// Mitsubishi GX Works2 project: Final_Version   PLC: FX3G

// global labels: Global1
VAR_GLOBAL
  DayStartSwitch AT X007 : BOOL;
  NotInStockSwitch AT M41 : BOOL;
  DayLight AT Y007 : BOOL;
  IceMakeSwitch AT X001 : BOOL;
  AnalogInput1 AT D8280 : INT;
END_VAR
VAR_GLOBAL CONSTANT
  UpperBound_K10 : REAL := 10.0;
  LowerBound_K0 : REAL;
  PetelNeeded_K280 : REAL := 280.0;
  LemonNeeded_K455 : REAL := 455.0;
  StabilityNeeded_K105 : REAL := 105.0;
  GumiBearsNeeded_K28 : REAL := 28.0;
  PetelNeeded_K385 : REAL := 385.0;
  LemonNeeded_K665 : REAL := 665.0;
  StabilityNeeded_K210 : REAL := 210.0;
  GumiBearsNeeded_K70 : REAL := 70.0;
END_VAR
VAR_GLOBAL
  RegularGumiLight AT M42 : BOOL;
END_VAR
VAR_GLOBAL CONSTANT
  Regular_GumiGam_k5 : REAL := 5.0;
  Special_GumiGam_K6 : REAL := 6.0;
END_VAR
VAR_GLOBAL
  IceMakeLight AT Y000 : BOOL;
  IceMakeTimer AT TC1 : BOOL;
  DayFinishSwitch AT M11 : BOOL;
END_VAR
VAR_GLOBAL CONSTANT
  IceMakeCounter_K50 : INT := 50;
  CounterValue_K1 : INT := 1;
  K400_const : REAL := 400.0;
END_VAR
VAR_GLOBAL
  PossibleRegularGumi AT M43 : BOOL;
  SpecialGumiLight AT M45 : BOOL;
  IcePetelContainer_IceMake AT D1500 : REAL;
  IceLemonContainer_IceMake AT D2500 : REAL;
  SaveAnalog_1_Value AT D5100 : REAL;
  PetelStock AT D1100 : REAL;
  LemonStock AT D2100 : REAL;
  StabilityStock AT D3100 : REAL;
  GumiBearsStock AT D4100 : REAL;
  IceMakeCounter_Finish AT CS0 : BOOL;
  IceMakeTimer_Finish AT TS1 : BOOL;
  IceMakeCounter AT CC0 : BOOL;
END_VAR
VAR_GLOBAL CONSTANT
  IceMakeTimer_K50 : INT := 50;
END_VAR
VAR_GLOBAL
  PossibleSpecialGumi AT M44 : BOOL;
  CoolingSwitchX002 AT X002 : BOOL;
  CoolingContainerPetel AT D6000 : REAL;
  CoolingContainerLemon AT D6010 : REAL;
  CoolingTimerDone AT TS2 : BOOL;
  CoolingFinishedCounter AT CC7 : BOOL;
  CoolingLightY002 AT Y002 : BOOL;
  CoolingTimer AT TC2 : BOOL;
END_VAR
VAR_GLOBAL CONSTANT
  CoolingTimeValue : INT := 80;
END_VAR
VAR_GLOBAL
  TempIndicatorX003 AT X003 : BOOL;
END_VAR
VAR_GLOBAL CONSTANT
  NormalGumiBears : REAL := 28;
  PinukGumiBears : REAL := 70;
  ResetContainer : REAL;
END_VAR
VAR_GLOBAL
  MixingContainer AT D6030 : REAL;
END_VAR
VAR_GLOBAL CONSTANT
  BlinkingCounterNormal : REAL := 3;
END_VAR
VAR_GLOBAL
  BlinkingCounterChosen AT D6040 : REAL;
END_VAR
VAR_GLOBAL CONSTANT
  BlinkingCounterPinuk : REAL := 5;
END_VAR
VAR_GLOBAL
  BlinkingLight5 AT Y005 : BOOL;
END_VAR
VAR_GLOBAL CONSTANT
  BlinkingTimerValue : INT := 10;
END_VAR
VAR_GLOBAL
  BlinkingTimer1 AT TC24 : BOOL;
  blinkingTriger AT M32 : BOOL;
  BlinkingTimerDone1 AT TS24 : BOOL;
  BlinkingTimeIsUp AT CS10 : BOOL;
  BlinkingLight6 AT Y006 : BOOL;
  BlinkingTimer2 AT TC25 : BOOL;
  BlinkingTimerDone2 AT TS25 : BOOL;
  BlinkingTimesUpCounter AT CC10 : BOOL;
  Stock AT D6050 : REAL;
END_VAR
VAR_GLOBAL CONSTANT
  FinishedPackage : REAL := 1;
END_VAR
VAR_GLOBAL
  AnalogOut AT D8282 : INT;
  EmergencyStop AT X005 : BOOL;
END_VAR
VAR_GLOBAL CONSTANT
  K40_const : REAL := 40;
  IcePetelRegular_K350 : REAL := 350;
  IcePetelPinuk_K560 : REAL := 560;
  IceLemonRegular_K490 : REAL := 490;
  IceLemonPinuk_K700 : REAL := 700;
END_VAR
VAR_GLOBAL
  InValidInput AT Y010 : BOOL;
  CoolingFinishedCounter_Finish AT CS7 : BOOL;
END_VAR

// task Task_01 (event TRUE, interval 0, priority 31): POU_01

PROGRAM POU_01
(* structured ladder/FBD written out as ST: instructions are called as NAME(EN, inputs, outputs); _pN, _eN, _tN stand for wires *)
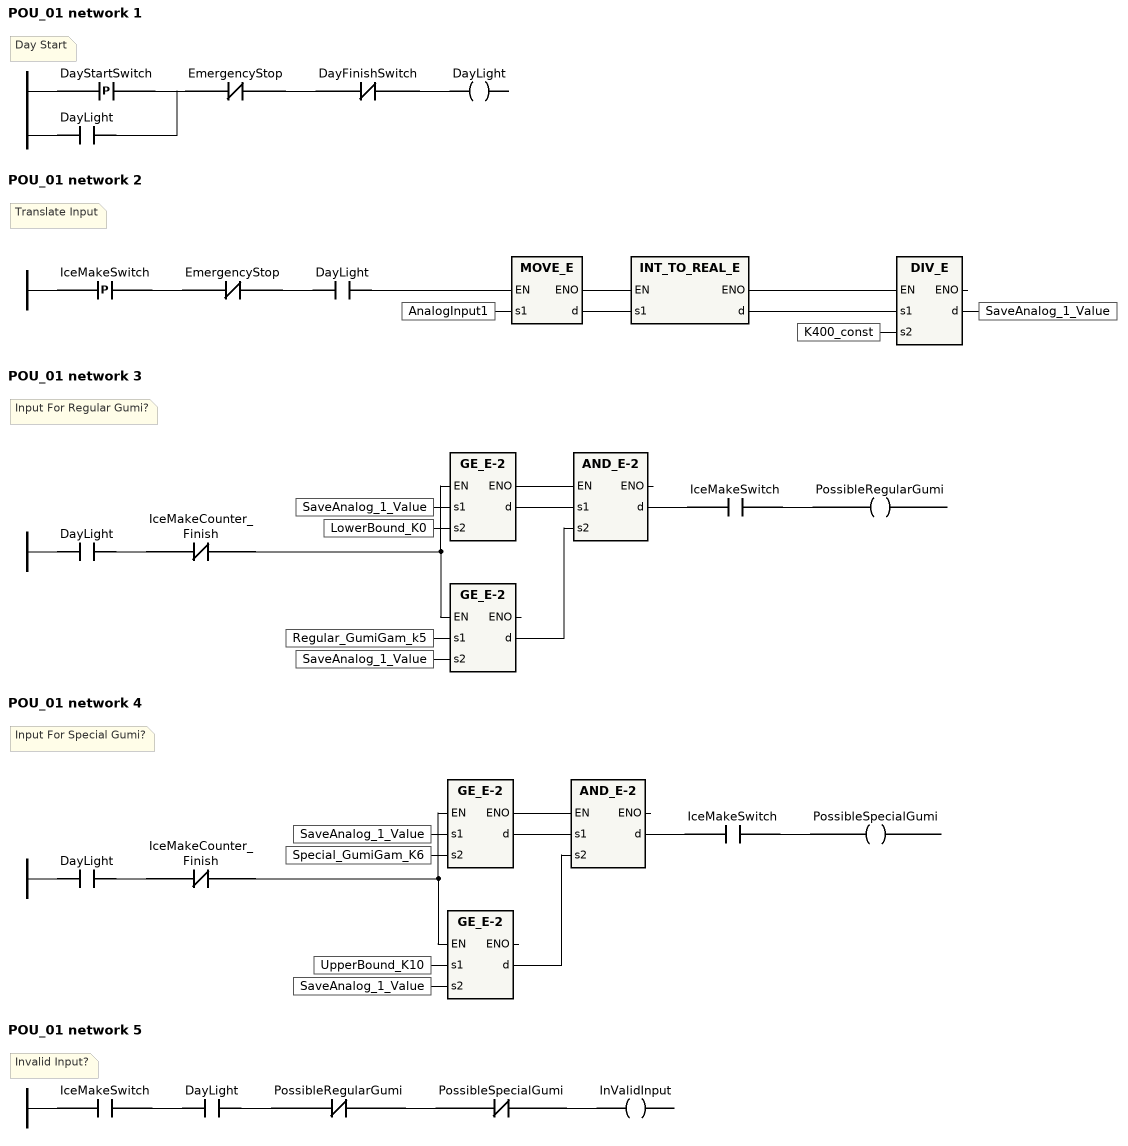
(* network 1 *)
(* Day Start *)
DayLight := ((LDP(TRUE, DayStartSwitch) OR DayLight) AND NOT EmergencyStop) AND NOT DayFinishSwitch;
(* network 2 *)
(* Translate Input *)
_e2 := MOVE_E(LDP(TRUE, IceMakeSwitch) AND NOT EmergencyStop AND DayLight, AnalogInput1, _t1);
_e4 := INT_TO_REAL_E(_e2, _t1, _t3);
DIV_E(_e4, _t3, K400_const, SaveAnalog_1_Value);
(* network 3 *)
(* Input For Regular Gumi? *)
_p1 := DayLight AND NOT IceMakeCounter_Finish;
_e3 := GE_E(_p1, SaveAnalog_1_Value, LowerBound_K0, _t2);
GE_E(_p1, Regular_GumiGam_k5, SaveAnalog_1_Value, _t4);
AND_E(_e3, _t2, _t4, _t5);
PossibleRegularGumi := _t5 AND IceMakeSwitch;
(* network 4 *)
(* Input For Special Gumi? *)
_p1 := DayLight AND NOT IceMakeCounter_Finish;
_e3 := GE_E(_p1, SaveAnalog_1_Value, Special_GumiGam_K6, _t2);
GE_E(_p1, UpperBound_K10, SaveAnalog_1_Value, _t4);
AND_E(_e3, _t2, _t4, _t5);
PossibleSpecialGumi := _t5 AND IceMakeSwitch;
(* network 5 *)
(* Invalid Input? *)
InValidInput := IceMakeSwitch AND DayLight AND NOT PossibleRegularGumi AND NOT PossibleSpecialGumi;
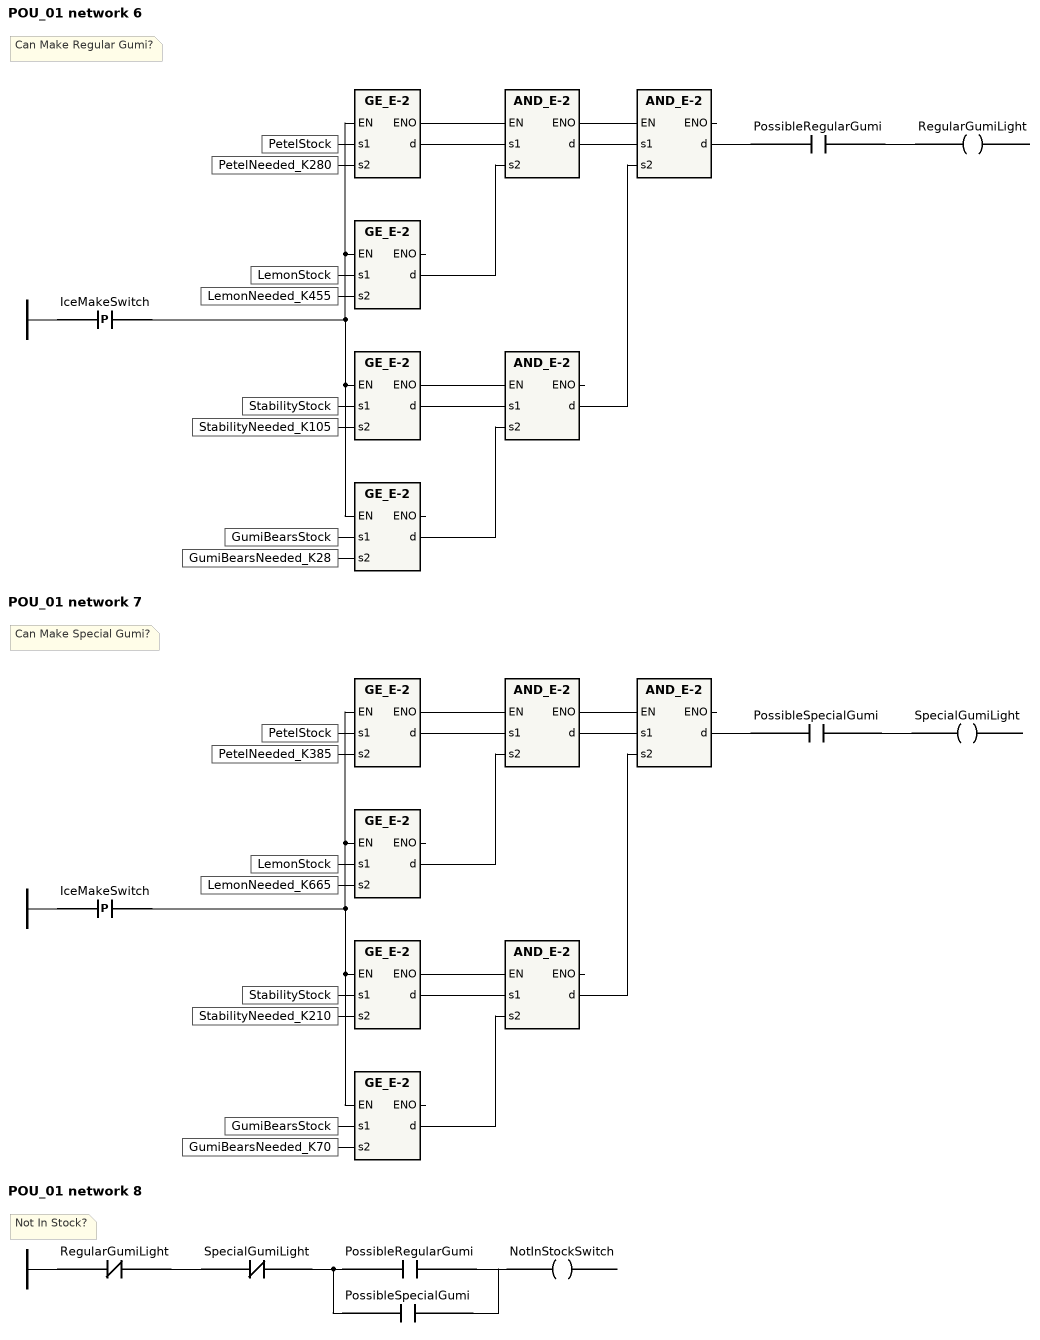
(* network 6 *)
(* Can Make Regular Gumi? *)
_p1 := LDP(TRUE, IceMakeSwitch);
_e3 := GE_E(_p1, PetelStock, PetelNeeded_K280, _t2);
GE_E(_p1, LemonStock, LemonNeeded_K455, _t4);
_e6 := AND_E(_e3, _t2, _t4, _t5);
_e8 := GE_E(_p1, StabilityStock, StabilityNeeded_K105, _t7);
GE_E(_p1, GumiBearsStock, GumiBearsNeeded_K28, _t9);
AND_E(_e8, _t7, _t9, _t10);
AND_E(_e6, _t5, _t10, _t11);
RegularGumiLight := _t11 AND PossibleRegularGumi;
(* network 7 *)
(* Can Make Special Gumi? *)
_p1 := LDP(TRUE, IceMakeSwitch);
_e3 := GE_E(_p1, PetelStock, PetelNeeded_K385, _t2);
GE_E(_p1, LemonStock, LemonNeeded_K665, _t4);
_e6 := AND_E(_e3, _t2, _t4, _t5);
_e8 := GE_E(_p1, StabilityStock, StabilityNeeded_K210, _t7);
GE_E(_p1, GumiBearsStock, GumiBearsNeeded_K70, _t9);
AND_E(_e8, _t7, _t9, _t10);
AND_E(_e6, _t5, _t10, _t11);
SpecialGumiLight := _t11 AND PossibleSpecialGumi;
(* network 8 *)
(* Not In Stock? *)
_p1 := NOT RegularGumiLight AND NOT SpecialGumiLight;
NotInStockSwitch := (_p1 AND PossibleRegularGumi) OR (_p1 AND PossibleSpecialGumi);
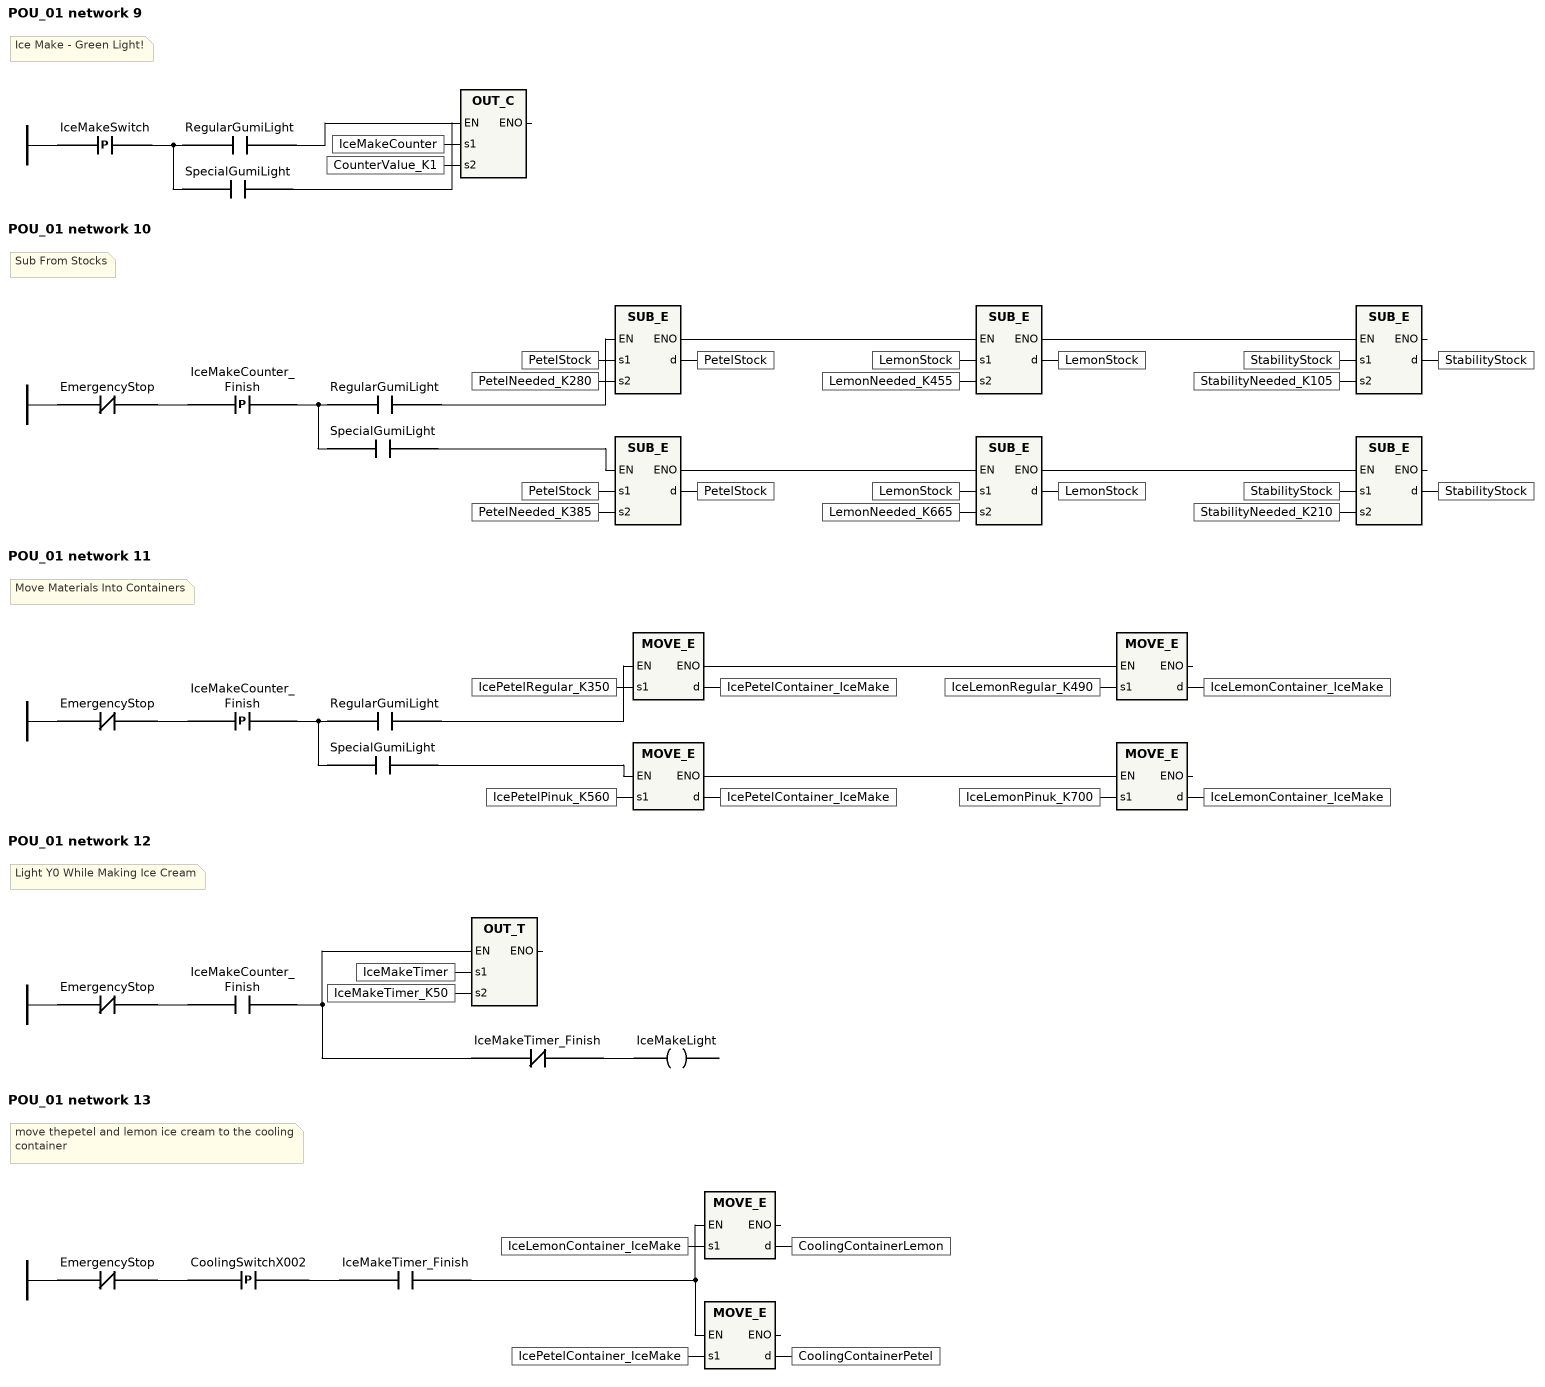
(* network 9 *)
(* Ice Make - Green Light! *)
_p1 := LDP(TRUE, IceMakeSwitch);
OUT_C((_p1 AND RegularGumiLight) OR (_p1 AND SpecialGumiLight), IceMakeCounter, CounterValue_K1);
(* network 10 *)
(* Sub From Stocks *)
_p1 := NOT EmergencyStop AND LDP(TRUE, IceMakeCounter_Finish);
_e2 := SUB_E(_p1 AND RegularGumiLight, PetelStock, PetelNeeded_K280, PetelStock);
_e3 := SUB_E(_e2, LemonStock, LemonNeeded_K455, LemonStock);
SUB_E(_e3, StabilityStock, StabilityNeeded_K105, StabilityStock);
_e4 := SUB_E(_p1 AND SpecialGumiLight, PetelStock, PetelNeeded_K385, PetelStock);
_e5 := SUB_E(_e4, LemonStock, LemonNeeded_K665, LemonStock);
SUB_E(_e5, StabilityStock, StabilityNeeded_K210, StabilityStock);
(* network 11 *)
(* Move Materials Into Containers *)
_p1 := NOT EmergencyStop AND LDP(TRUE, IceMakeCounter_Finish);
_e2 := MOVE_E(_p1 AND RegularGumiLight, IcePetelRegular_K350, IcePetelContainer_IceMake);
MOVE_E(_e2, IceLemonRegular_K490, IceLemonContainer_IceMake);
_e3 := MOVE_E(_p1 AND SpecialGumiLight, IcePetelPinuk_K560, IcePetelContainer_IceMake);
MOVE_E(_e3, IceLemonPinuk_K700, IceLemonContainer_IceMake);
(* network 12 *)
(* Light Y0 While Making Ice Cream *)
_p1 := NOT EmergencyStop AND IceMakeCounter_Finish;
OUT_T(_p1, IceMakeTimer, IceMakeTimer_K50);
IceMakeLight := _p1 AND NOT IceMakeTimer_Finish;
(* network 13 *)
(* move thepetel and lemon ice cream to the cooling container *)
_p1 := NOT EmergencyStop AND LDP(TRUE, CoolingSwitchX002) AND IceMakeTimer_Finish;
MOVE_E(_p1, IceLemonContainer_IceMake, CoolingContainerLemon);
MOVE_E(_p1, IcePetelContainer_IceMake, CoolingContainerPetel);
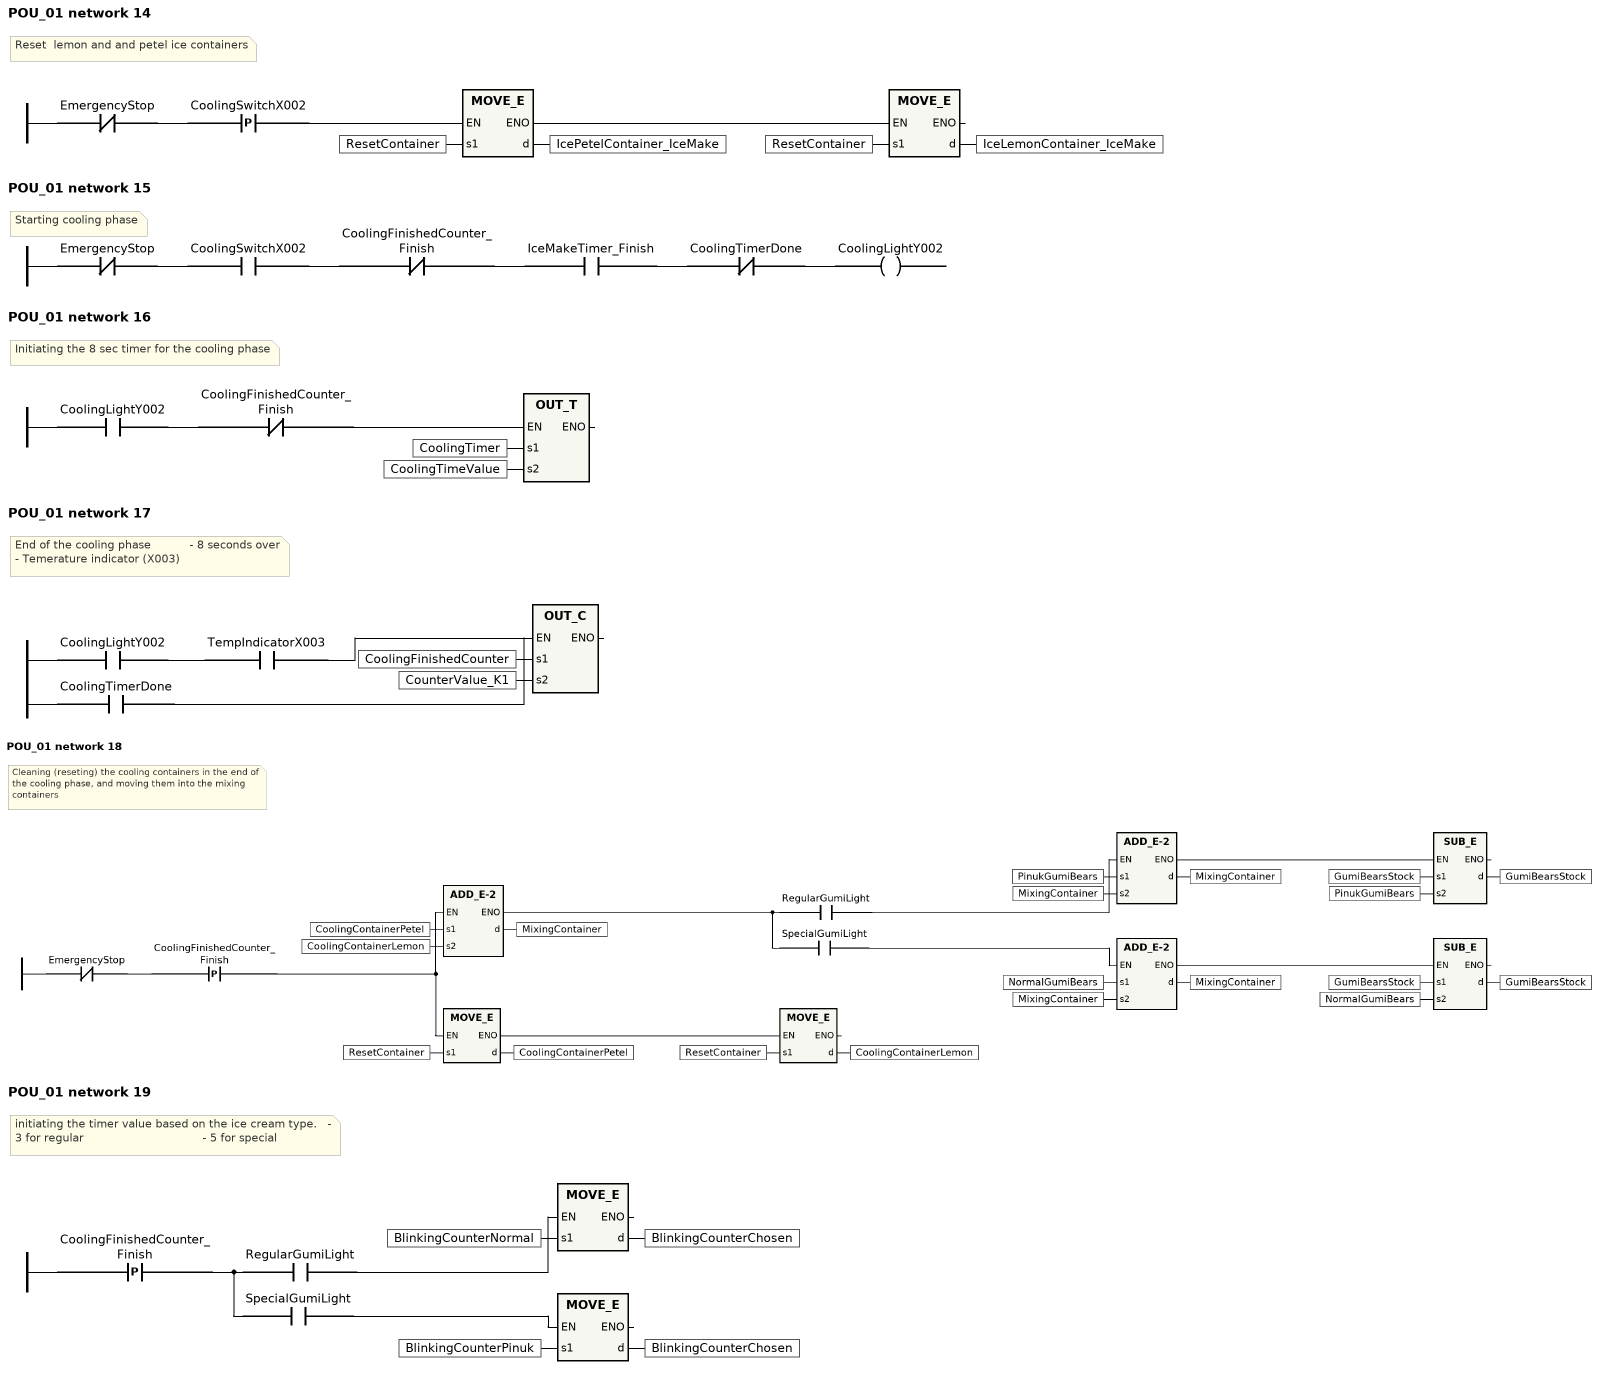
(* network 14 *)
(* Reset  lemon and and petel ice containers *)
_e1 := MOVE_E(NOT EmergencyStop AND LDP(TRUE, CoolingSwitchX002), ResetContainer, IcePetelContainer_IceMake);
MOVE_E(_e1, ResetContainer, IceLemonContainer_IceMake);
(* network 15 *)
(* Starting cooling phase *)
CoolingLightY002 := NOT EmergencyStop AND CoolingSwitchX002 AND NOT CoolingFinishedCounter_Finish AND IceMakeTimer_Finish AND NOT CoolingTimerDone;
(* network 16 *)
(* Initiating the 8 sec timer for the cooling phase *)
OUT_T(CoolingLightY002 AND NOT CoolingFinishedCounter_Finish, CoolingTimer, CoolingTimeValue);
(* network 17 *)
(* End of the cooling phase           - 8 seconds over                          - Temerature indicator (X003) *)
OUT_C((CoolingLightY002 AND TempIndicatorX003) OR CoolingTimerDone, CoolingFinishedCounter, CounterValue_K1);
(* network 18 *)
(* Cleaning (reseting) the cooling containers in the end of the cooling phase, and moving them into the mixing containers *)
_p1 := NOT EmergencyStop AND LDP(TRUE, CoolingFinishedCounter_Finish);
_e2 := ADD_E(_p1, CoolingContainerPetel, CoolingContainerLemon, MixingContainer);
_e3 := ADD_E(_e2 AND RegularGumiLight, PinukGumiBears, MixingContainer, MixingContainer);
SUB_E(_e3, GumiBearsStock, PinukGumiBears, GumiBearsStock);
_e4 := ADD_E(_e2 AND SpecialGumiLight, NormalGumiBears, MixingContainer, MixingContainer);
SUB_E(_e4, GumiBearsStock, NormalGumiBears, GumiBearsStock);
_e5 := MOVE_E(_p1, ResetContainer, CoolingContainerPetel);
MOVE_E(_e5, ResetContainer, CoolingContainerLemon);
(* network 19 *)
(* initiating the timer value based on the ice cream type.   - 3 for regular                                  - 5 for special *)
_p1 := LDP(TRUE, CoolingFinishedCounter_Finish);
MOVE_E(_p1 AND RegularGumiLight, BlinkingCounterNormal, BlinkingCounterChosen);
MOVE_E(_p1 AND SpecialGumiLight, BlinkingCounterPinuk, BlinkingCounterChosen);
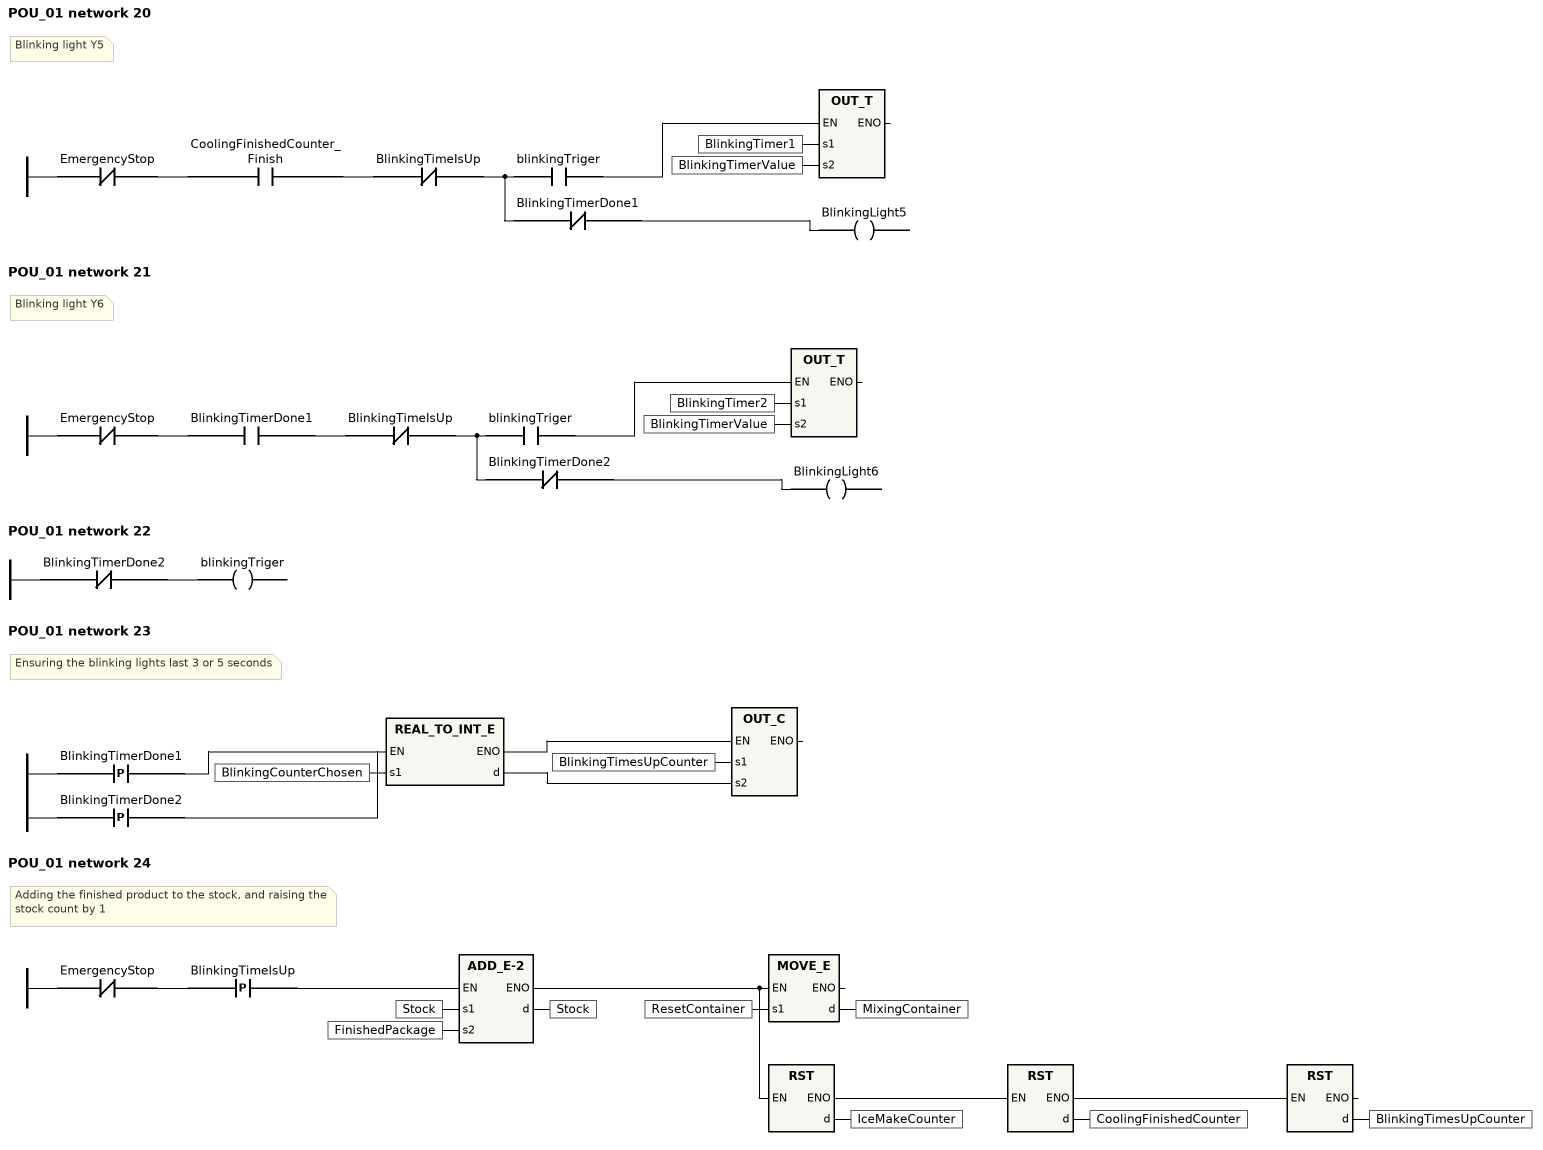
(* network 20 *)
(* Blinking light Y5 *)
_p1 := NOT EmergencyStop AND CoolingFinishedCounter_Finish AND NOT BlinkingTimeIsUp;
OUT_T(_p1 AND blinkingTriger, BlinkingTimer1, BlinkingTimerValue);
BlinkingLight5 := _p1 AND NOT BlinkingTimerDone1;
(* network 21 *)
(* Blinking light Y6 *)
_p1 := NOT EmergencyStop AND BlinkingTimerDone1 AND NOT BlinkingTimeIsUp;
OUT_T(_p1 AND blinkingTriger, BlinkingTimer2, BlinkingTimerValue);
BlinkingLight6 := _p1 AND NOT BlinkingTimerDone2;
(* network 22 *)
blinkingTriger := NOT BlinkingTimerDone2;
(* network 23 *)
(* Ensuring the blinking lights last 3 or 5 seconds *)
_e2 := REAL_TO_INT_E(LDP(TRUE, BlinkingTimerDone1) OR LDP(TRUE, BlinkingTimerDone2), BlinkingCounterChosen, _t1);
OUT_C(_e2, BlinkingTimesUpCounter, _t1);
(* network 24 *)
(* Adding the finished product to the stock, and raising the stock count by 1 *)
_e1 := ADD_E(NOT EmergencyStop AND LDP(TRUE, BlinkingTimeIsUp), Stock, FinishedPackage, Stock);
MOVE_E(_e1, ResetContainer, MixingContainer);
_e2 := RST(_e1, IceMakeCounter);
_e3 := RST(_e2, CoolingFinishedCounter);
RST(_e3, BlinkingTimesUpCounter);
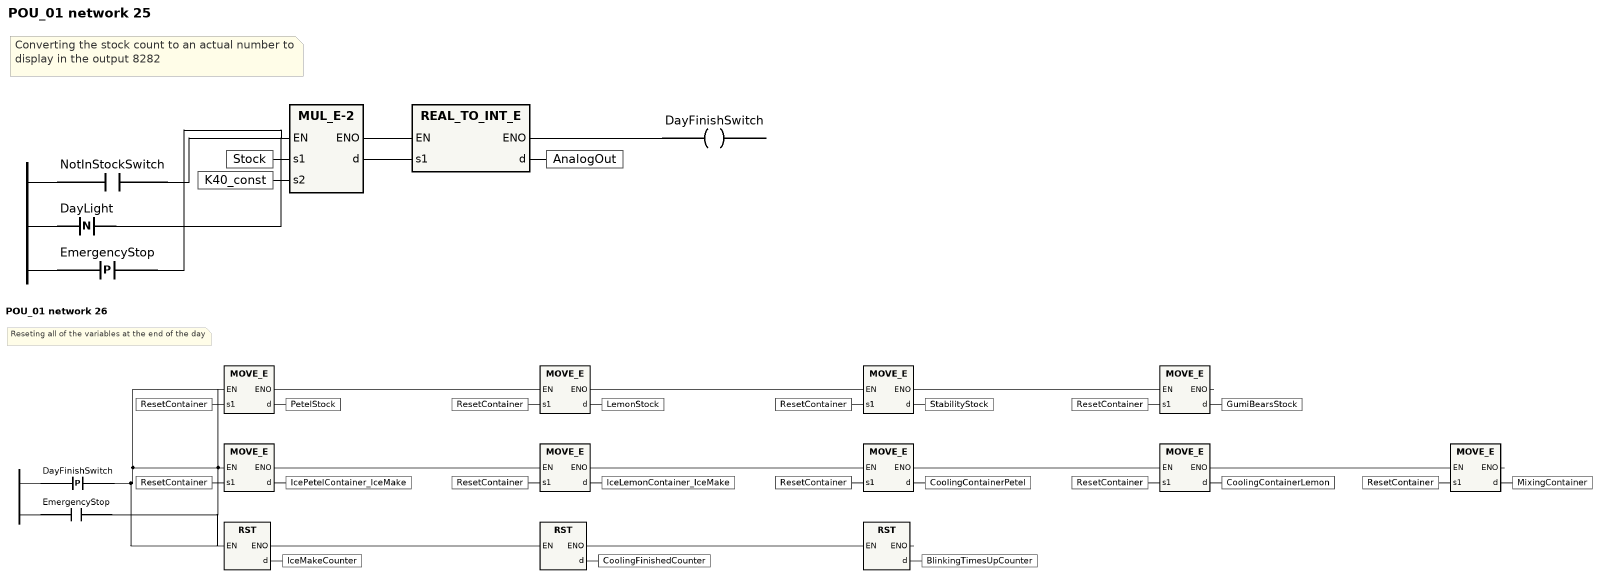
(* network 25 *)
(* Converting the stock count to an actual number to display in the output 8282 *)
_e2 := MUL_E(NotInStockSwitch OR LDF(TRUE, DayLight) OR LDP(TRUE, EmergencyStop), Stock, K40_const, _t1);
_e3 := REAL_TO_INT_E(_e2, _t1, AnalogOut);
DayFinishSwitch := _e3;
(* network 26 *)
(* Reseting all of the variables at the end of the day *)
_p1 := LDP(TRUE, DayFinishSwitch) OR EmergencyStop;
_e2 := MOVE_E(_p1, ResetContainer, PetelStock);
_e3 := MOVE_E(_e2, ResetContainer, LemonStock);
_e4 := MOVE_E(_e3, ResetContainer, StabilityStock);
MOVE_E(_e4, ResetContainer, GumiBearsStock);
_e5 := MOVE_E(_p1, ResetContainer, IcePetelContainer_IceMake);
_e6 := MOVE_E(_e5, ResetContainer, IceLemonContainer_IceMake);
_e7 := MOVE_E(_e6, ResetContainer, CoolingContainerPetel);
_e8 := MOVE_E(_e7, ResetContainer, CoolingContainerLemon);
MOVE_E(_e8, ResetContainer, MixingContainer);
_e9 := RST(_p1, IceMakeCounter);
_e10 := RST(_e9, CoolingFinishedCounter);
RST(_e10, BlinkingTimesUpCounter);
END_PROGRAM
